// TIA Portal V19 program export: 1 tag tables, 0 data types, 0 data blocks, 1 code blocks (in call order from the OBs), 0 instance data blocks

VAR_GLOBAL   // PLC tag table "Standard-Variablentabelle"
   start AT %I0.0 : Bool;
   motor AT %Q0.0 : Bool;
   stop AT %I0.1 : Bool;
   mem AT %M0.2 : Bool;
END_VAR

ORGANIZATION_BLOCK "Main"   // OB1, LAD, ProgramCycle
TITLE = "Main Program Sweep (Cycle)"
{ S7_Optimized_Access := 'TRUE' }
// stored: SetENOAutomatically false
   VAR_INPUT
      Initial_Call : Bool;   // Initial call of this OB
      Remanence : Bool;   // =True, if remanent data are available
   END_VAR
BEGIN

REGION Network 1
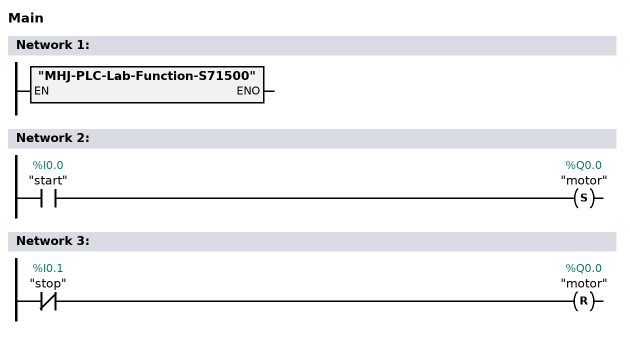
   RUNG wire#powerrail
      "MHJ-PLC-Lab-Function-S71500"()
   END_RUNG
   // the same network as SCL:
   "MHJ-PLC-Lab-Function-S71500"();
END_REGION

REGION Network 2
   RUNG wire#powerrail
      Contact( "start" )
      S_Coil( "motor" )
   END_RUNG
   // the same network as SCL:
   IF "start" THEN "motor" := TRUE; END_IF;
END_REGION

REGION Network 3
   RUNG wire#powerrail
      I_Contact( "stop" )
      R_Coil( "motor" )
   END_RUNG
   // the same network as SCL:
   IF NOT "stop" THEN "motor" := FALSE; END_IF;
END_REGION
END_ORGANIZATION_BLOCK
